Staubli VAL3: decSetDrvPwrMsg.pgx

public program decSetDrvPwrMsg(bool& x_bFlag (dimensions=1))
  local num l_nData
  local num l_nIndex
  local num l_nRetVal
begin
  // Copyright (c) 2021, Institute for Factory Automation and Production Systems (FAPS)
  //
  // Licensed under the Apache License, Version 2.0 (the "License");
  // you may not use this file except in compliance with the License.
  // You may obtain a copy of the License at
  //
  //     http://www.apache.org/licenses/LICENSE-2.0
  //
  // Unless required by applicable law or agreed to in writing, software
  // distributed under the License is distributed on an "AS IS" BASIS,
  // WITHOUT WARRANTIES OR CONDITIONS OF ANY KIND, either express or implied.
  // See the License for the specific language governing permissions and
  // limitations under the License.


  // decode set drive power message body (data)

  // assume failure to decode
  setDrvPwrAck.header.nReplyCode=SimpleMsg:ReplyCode.FAILURE

  // fields:
  //  setDrvPwrMsg.bDrivePower


  // drive power, 1 byte
  l_nRetVal=fromBinary(setDrvPwrMsg.body.nData,1,"1",l_nData)

  if (l_nRetVal!=1)
    x_bFlag=false
    return
  endIf

  if (l_nData==1)
    setDrvPwrMsg.bDrivePower=true
  elseIf (l_nData==0)
    setDrvPwrMsg.bDrivePower=false
  else
    // TODO: debug output
    x_bFlag=false
    return
  endIf

  // decoding successful
  setDrvPwrAck.header.nReplyCode=SimpleMsg:ReplyCode.SUCCESS
  x_bFlag=true
end
